PROGRAM MAIN
VAR
	//Conveyor
	Conveyor		: FB_Conveyor;
	
	// Station 1
	Station1_Bin1	: FB_StationBin;
	Station1_Bin2	: FB_StationBin;
	Station1_Bin3	: FB_StationBin;
	
	//Station 2
	Station2_Bin1	: FB_StationBin;
	Station2_Bin2	: FB_StationBin;
	Station2_Bin3	: FB_StationBin;
	
	// Stations Ready
	bStation1_Ready : BOOL;
	bStation2_Ready : BOOL;
	
	// Reset Bins
	bResetCount_Bin1: BOOL;
	bResetCount_Bin2: BOOL;
	bResetCount_Bin3: BOOL;
	bResetCount_Bin4: BOOL;
	bResetCount_Bin5: BOOL;
	bResetCount_Bin6: BOOL;
END_VAR

a_EnableDrives();

Conveyor(
	Station_1_Ready:= bStation1_Ready, 
	Station_2_Ready:= bStation2_Ready, 
	At_Station_1=> , 
	At_Station_2=> , 
	At_Station_3=> , 
	ResetConvoyor := Globals.ConveyorControl.bReset,
	sStatus=> Globals.ConveyorControl.sStatus, 
	bError=> Globals.ConveyorControl.bError);
	
Station1_Bin1(
	bEnableBin := Globals.Bin1Control.bEnable,
	Home_Sensor:= IO.iStation_1_1_Home_Sensor, 
	Safe_Sensor:= IO.iStation_1_1_Safe_Sensor, 
	Dispense_Sensor:= IO.iStation_1_1_Dispense_Sensor, 
	Part_Present := IO.iStation_1_1_Part_Present_Sensor,
	Dependency_OK:= NOT Station1_Bin2.Lock_Dependency AND NOT Station1_Bin3.Lock_Dependency, 
	At_Station:= Conveyor.At_Station_1, 
	Trigger_OF_Drive=> IO.oR1_NO_Contact, 
	Direction_OF_Drive=> IO.oDirection_OF_Driver_1, 
	Lock_Dependency=> , 
	ResetPartCount := bResetCount_Bin1,
	ResetBin := Globals.Bin1Control.bReset,
	bError=> Globals.Bin1Control.bError, 
	sStatus=> Globals.Bin1Control.sStatus);
	
Station1_Bin2(
	bEnableBin := Globals.Bin2Control.bEnable,
	Home_Sensor:= IO.iStation_1_2_Home_Sensor, 
	Safe_Sensor:= IO.iStation_1_2_Safe_Sensor, 
	Dispense_Sensor:= IO.iStation_1_2_Dispense_Sensor,
	Part_Present := IO.iStation_1_2_Part_Present_Sensor, 
	Dependency_OK:= NOT Station1_Bin1.Lock_Dependency AND NOT Station1_Bin3.Lock_Dependency, 
	At_Station:= Conveyor.At_Station_1, 
	Trigger_OF_Drive=> IO.oR2_NO_Contact, 
	Direction_OF_Drive=> IO.oDirection_OF_Driver_2, 
	Lock_Dependency=> , 
	ResetPartCount := bResetCount_Bin2,
	ResetBin := Globals.Bin2Control.bReset,
	bError=> Globals.Bin2Control.bError , 
	sStatus=> Globals.Bin2Control.sStatus);
	
Station1_Bin3(
	bEnableBin := Globals.Bin3Control.bEnable,
	Home_Sensor:= IO.iStation_1_3_Home_Sensor, 
	Safe_Sensor:= IO.iStation_1_3_Safe_Sensor, 
	Dispense_Sensor:= IO.iStation_1_3_Dispense_Sensor,
	Part_Present := IO.iStation_1_3_Part_Present_Sensor, 
	Dependency_OK:= NOT Station1_Bin1.Lock_Dependency AND NOT Station1_Bin2.Lock_Dependency, 
	At_Station:= Conveyor.At_Station_1, 
	Trigger_OF_Drive=> IO.oR3_NO_Contact, 
	Direction_OF_Drive=> IO.oDirection_OF_Driver_3, 
	Lock_Dependency=> , 
	ResetPartCount := bResetCount_Bin3,
	ResetBin := Globals.Bin3Control.bReset,
	bError=> Globals.Bin3Control.bError, 
	sStatus=> Globals.Bin3Control.sStatus);
	
Station2_Bin1(
	bEnableBin := Globals.Bin4Control.bEnable,
	Home_Sensor:= IO.iStation_2_1_Home_Sensor, 
	Safe_Sensor:= IO.iStation_2_1_Safe_Sensor, 
	Dispense_Sensor:= IO.iStation_2_1_Dispense_Sensor,
	Part_Present := IO.iStation_2_1_Part_Present_Sensor, 
	Dependency_OK:= NOT Station2_Bin2.Lock_Dependency AND NOT Station2_Bin3.Lock_Dependency, 
	At_Station:= Conveyor.At_Station_2, 
	Trigger_OF_Drive=> IO.oR4_NO_Contact, 
	Direction_OF_Drive=> IO.oDirection_OF_Driver_4, 
	Lock_Dependency=> , 
	ResetPartCount := bResetCount_Bin4,
	ResetBin := Globals.Bin4Control.bReset,
	bError=>Globals.Bin4Control.bError , 
	sStatus=> Globals.Bin4Control.sStatus);
	
Station2_Bin2(
	bEnableBin := Globals.Bin5Control.bEnable,
	Home_Sensor:= IO.iStation_2_2_Home_Sensor, 
	Safe_Sensor:= IO.iStation_2_2_Safe_Sensor, 
	Dispense_Sensor:= IO.iStation_2_2_Dispense_Sensor, 
	Part_Present := IO.iStation_2_2_Part_Present_Sensor,
	Dependency_OK:= NOT Station2_Bin1.Lock_Dependency AND NOT Station2_Bin3.Lock_Dependency, 
	At_Station:= Conveyor.At_Station_2, 
	Trigger_OF_Drive=> IO.oR5_NO_Contact, 
	Direction_OF_Drive=> IO.oDirection_OF_Driver_5, 
	Lock_Dependency=> , 
	ResetPartCount := bResetCount_Bin5,
	ResetBin := Globals.Bin5Control.bReset,
	bError=> Globals.Bin5Control.bError, 
	sStatus=> Globals.Bin5Control.sStatus);
	
Station2_Bin3(
	bEnableBin := Globals.Bin6Control.bEnable,
	Home_Sensor:= IO.iStation_2_3_Home_Sensor, 
	Safe_Sensor:= IO.iStation_2_3_Safe_Sensor, 
	Dispense_Sensor:= IO.iStation_2_3_Dispense_Sensor,
	Part_Present := IO.iStation_2_3_Part_Present_Sensor, 
	Dependency_OK:= NOT Station2_Bin1.Lock_Dependency AND NOT Station2_Bin2.Lock_Dependency, 
	At_Station:= Conveyor.At_Station_2, 
	Trigger_OF_Drive=> IO.oR6_NO_Contact, 
	Direction_OF_Drive=> IO.oDirection_OF_Driver_6, 
	Lock_Dependency=> , 
	ResetPartCount := bResetCount_Bin6,
	ResetBin := Globals.Bin6Control.bReset,
	bError=> Globals.Bin6Control.bError, 
	sStatus=> Globals.Bin6Control.sStatus);
	
// Ready Conditions
bStation1_Ready := Station1_Bin1.Count_OF_Parts + Station1_Bin2.Count_OF_Parts + Station1_Bin3.Count_OF_Parts >= 15;
bStation2_Ready := Station2_Bin1.Count_OF_Parts + Station2_Bin2.Count_OF_Parts + Station2_Bin3.Count_OF_Parts >= 15;
IF Globals.bResetPartCount_Station1 
AND (Station1_Bin1.Count_OF_Parts + Station1_Bin2.Count_OF_Parts + Station1_Bin3.Count_OF_Parts > 0) THEN
	bResetCount_Bin1:= TRUE;
	bResetCount_Bin2:= TRUE;
	bResetCount_Bin3:= TRUE;
ELSE
	Globals.bResetPartCount_Station1 := FALSE;
END_IF

IF Globals.bResetPartCount_Station2 
AND (Station2_Bin1.Count_OF_Parts + Station2_Bin2.Count_OF_Parts + Station2_Bin3.Count_OF_Parts > 0) THEN
	bResetCount_Bin4 := TRUE;
	bResetCount_Bin5 := TRUE;
	bResetCount_Bin6 := TRUE;
ELSE
	Globals.bResetPartCount_Station2 := FALSE;
END_IF

ACTION a_EnableDrives:
IO.oEnable_of_Driver_1 := TRUE;
IO.oEnable_of_Driver_2 := TRUE;
IO.oEnable_of_Driver_3 := TRUE;
IO.oEnable_of_Driver_4 := TRUE;
IO.oEnable_of_Driver_5 := TRUE;
IO.oEnable_of_Driver_6 := TRUE;
IO.oEnable_of_Driver_7 := TRUE;
IO.oEnable_of_Driver_8 := TRUE;
END_ACTION

END_PROGRAM

(* stored: Version 1.1.0.1, ProductVersion 3.1.4024.9
   POU MAIN: Id {e47a8857-7317-4c59-bd0b-c9409bde97c2}, SpecialFunc None
   Action a_EnableDrives: Id {89d47b60-9f71-42a4-aad9-e4c22c66f4be} *)
